# EPICS substitutions: example/testURRobot/iocBoot/ioctestURRobot/substitutions/fb_epid.substitutions
# $Id$

file "$(OPTICS)/opticsApp/Db/fb_epid.db"
  {
    {
        P=testURRobot:epid1,
	IN=testURRobot:epid1:sim.VAL,
	OUT=testURRobot:epid1:sim.D,
	MODE=PID,
	CALC=A,
	PERMIT1="testURRobot:epid1:on.VAL",
	PERMIT2="",
	PERMIT3="",
	PERMIT4=""
    }
  }
